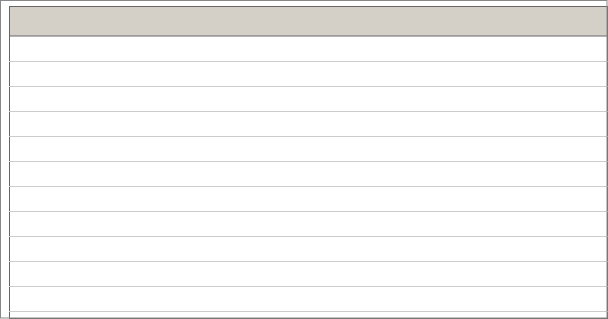
VISUALIZATION current  // 608x319
    Table (9,6 599x313), data array: MAIN.event_table_view.stAlarmEvents
        p3854506369: MAIN.event_table_view.stAlarmEvents[INDEX].nSourceId
        p1892666644: MAIN.event_table_view.stAlarmEvents[INDEX].nEventId
        p338671338: MAIN.event_table_view.stAlarmEvents[INDEX].Severity
        p2170511999: MAIN.event_table_view.stAlarmEvents[INDEX].ConfirmState
        p3723444502: MAIN.event_table_view.stAlarmEvents[INDEX].sDate
        p1218418051: MAIN.event_table_view.stAlarmEvents[INDEX].sTime
        p746581629: MAIN.event_table_view.stAlarmEvents[INDEX].Computer
        p3104783080: MAIN.event_table_view.stAlarmEvents[INDEX].sSource
        p2501879983: MAIN.event_table_view.stAlarmEvents[INDEX].MessageText
        p7306298: MAIN.event_table_view.stAlarmEvents[INDEX].bQuitMessage
        p1933151965: MAIN.event_table_view.stAlarmEvents[INDEX].bConfirmable
        p1755163831: 重要度
        p4092479075: 確認
        p2237128397: 日付
        p505689113: 時刻
        p2243050616: テキスト
END_VISUALIZATION

(* stored: Version 1.1.0.1, ProductVersion 3.1.4024.15
   Visu current: Id {2438d436-7f89-4bae-9c0b-71581f821792} *)
